(* Logix 5000 project; controller Uidaho_Factory vendor 1 type 14 code 165 rev 38.11; software revision 38.00; part 4 of 4 *)
(* tags used below, declared in another part *)
   MPO_Done : BOOL;
   MPO_Homing : BOOL;
   MPO_Oven_Start : BOOL;
   MPO_Turntable_Start : BOOL;
   SLD_Blue_Min : DINT;
   SLD_Blue_Time : DINT;
   SLD_Min_Value : DINT;
   SLD_Move_Time : DINT;
   SLD_Normal : DINT;
   SLD_Red_Min : DINT;
   SLD_Red_Time : DINT;
   SLD_start : DINT;
   SLD_Step : DINT;
   SLD_White_Time : DINT;
   Start : DINT;
   Step : DINT[20];
   StepTimers : TIMER[20];
   TurntableTimers : TIMER[10];
   VGR_HBW_Horizontal : DINT;   // The horizontal Encoder value for interfacing with HBW
   VGR_HBW_Rotate : DINT;
   VGR_HBW_Vertical : DINT;   // The Vertical Encoder value for interfacing with the HBW
   VGR_Horizontal_Target : DINT;
   VGR_Move_Horizontal : DINT;   // The horizontal encoder value for movement
   VGR_Move_Vertical : DINT;   // The vertical encoder value for movement
   VGR_MPO_Horizontal : DINT;   // The Horizontal encoderr value for interfacing with MPO
   VGR_MPO_Rotate : DINT;
   VGR_MPO_Vertical : DINT;   // The vertical encoder value for interfacing with MPO
   VGR_Rotation_Target : DINT;
   VGR_start : DINT;
   VGR_Step : DINT;
   VGR_Vertical_Target : DINT;
   Encoder_Counters_1X : COUNTER[10];
   PWM_Outputs : PWM_Out[20];
   Scaled_Analog_Color_Sensor_SLD : DINT;   // SLD - A1 = Color sensor
   VGR_PWM_Outputs : PWM_Out[20];
(* MainProgram, continued *)

ROUTINE MPO_Turntable_Process   (* ladder *)
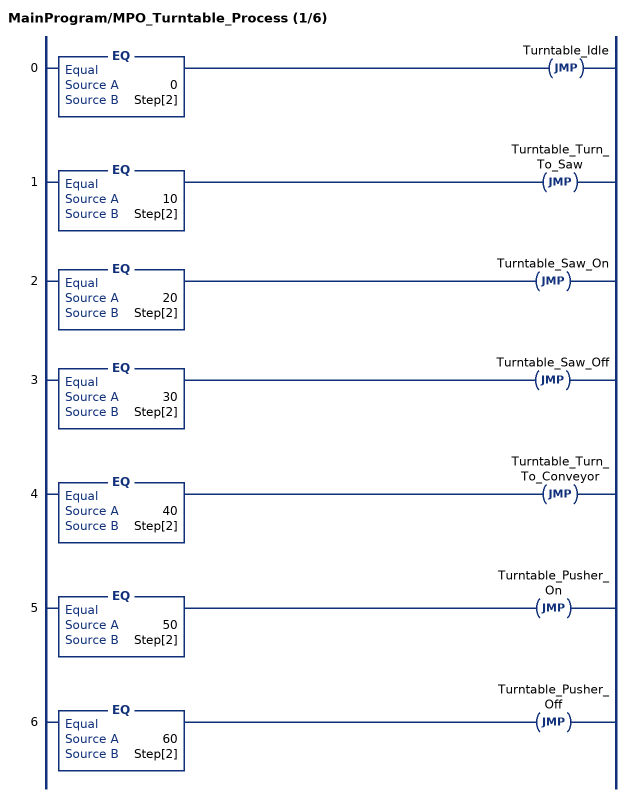
   0: EQ(0,Step[2])JMP(Turntable_Idle);
   1: EQ(10,Step[2])JMP(Turntable_Turn_To_Saw);
   2: EQ(20,Step[2])JMP(Turntable_Saw_On);
   3: EQ(30,Step[2])JMP(Turntable_Saw_Off);
   4: EQ(40,Step[2])JMP(Turntable_Turn_To_Conveyor);
   5: EQ(50,Step[2])JMP(Turntable_Pusher_On);
   6: EQ(60,Step[2])JMP(Turntable_Pusher_Off);
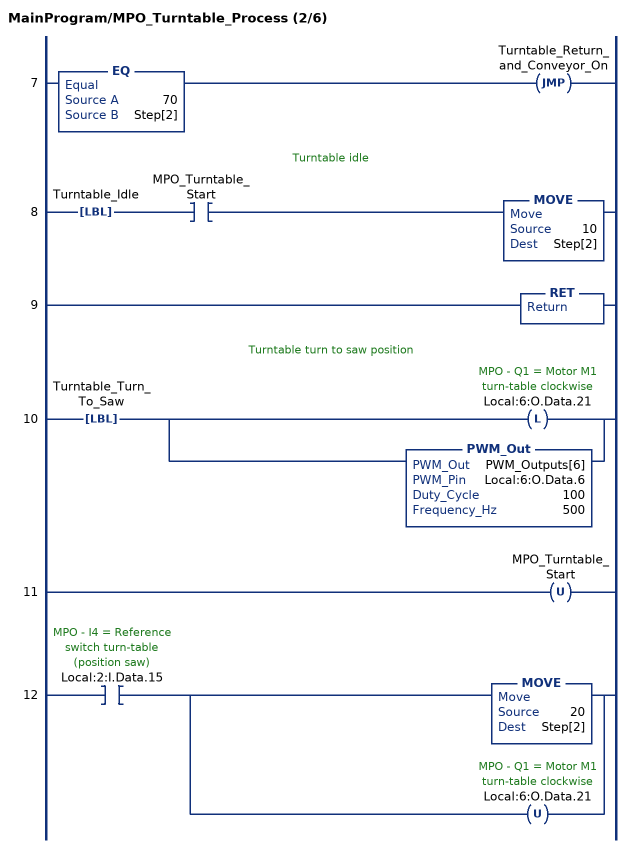
   7: EQ(70,Step[2])JMP(Turntable_Return_and_Conveyor_On);
   // Turntable idle
   8: LBL(Turntable_Idle)XIC(MPO_Turntable_Start)MOVE(10,Step[2]);
   9: RET();
   // Turntable turn to saw position
   10: LBL(Turntable_Turn_To_Saw)[OTL(Local:6:O.Data.21) ,PWM_Out(PWM_Outputs[6],Local:6:O.Data.6,100,500) ];
   11: OTU(MPO_Turntable_Start);
   12: XIC(Local:2:I.Data.15)[MOVE(20,Step[2]) ,OTU(Local:6:O.Data.21) ];
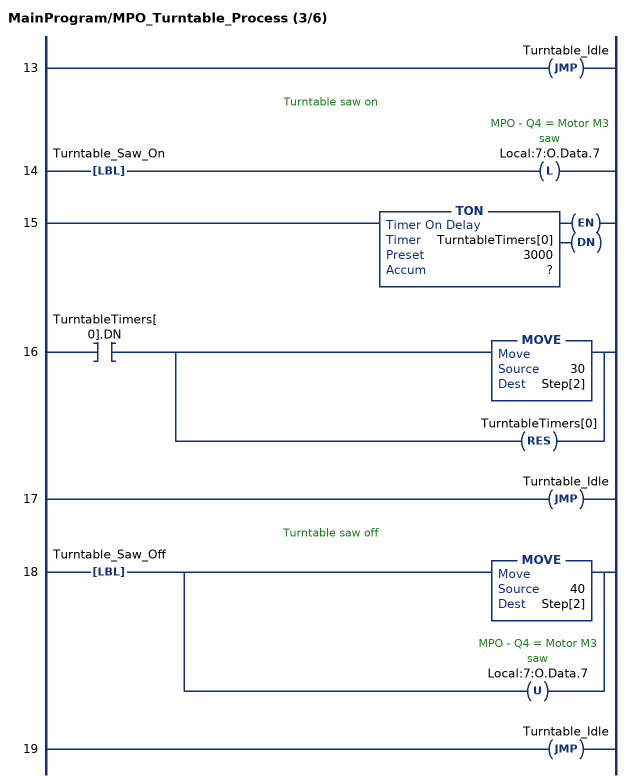
   13: JMP(Turntable_Idle);
   // Turntable saw on
   14: LBL(Turntable_Saw_On)OTL(Local:7:O.Data.7);
   15: TON(TurntableTimers[0],?,?);
   16: XIC(TurntableTimers[0].DN)[MOVE(30,Step[2]) ,RES(TurntableTimers[0]) ];
   17: JMP(Turntable_Idle);
   // Turntable saw off
   18: LBL(Turntable_Saw_Off)[MOVE(40,Step[2]) ,OTU(Local:7:O.Data.7) ];
   19: JMP(Turntable_Idle);
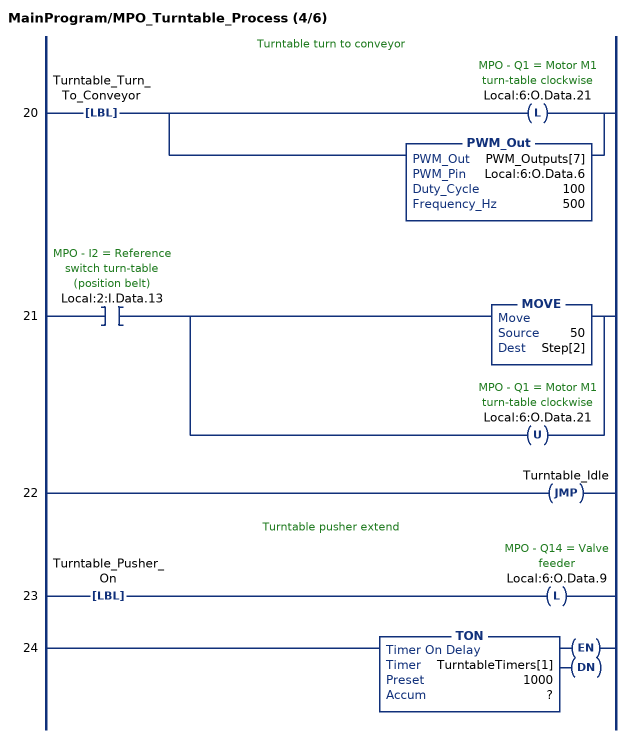
   // Turntable turn to conveyor
   20: LBL(Turntable_Turn_To_Conveyor)[OTL(Local:6:O.Data.21) ,PWM_Out(PWM_Outputs[7],Local:6:O.Data.6,100,500) ];
   21: XIC(Local:2:I.Data.13)[MOVE(50,Step[2]) ,OTU(Local:6:O.Data.21) ];
   22: JMP(Turntable_Idle);
   // Turntable pusher extend
   23: LBL(Turntable_Pusher_On)OTL(Local:6:O.Data.9);
   24: TON(TurntableTimers[1],?,?);
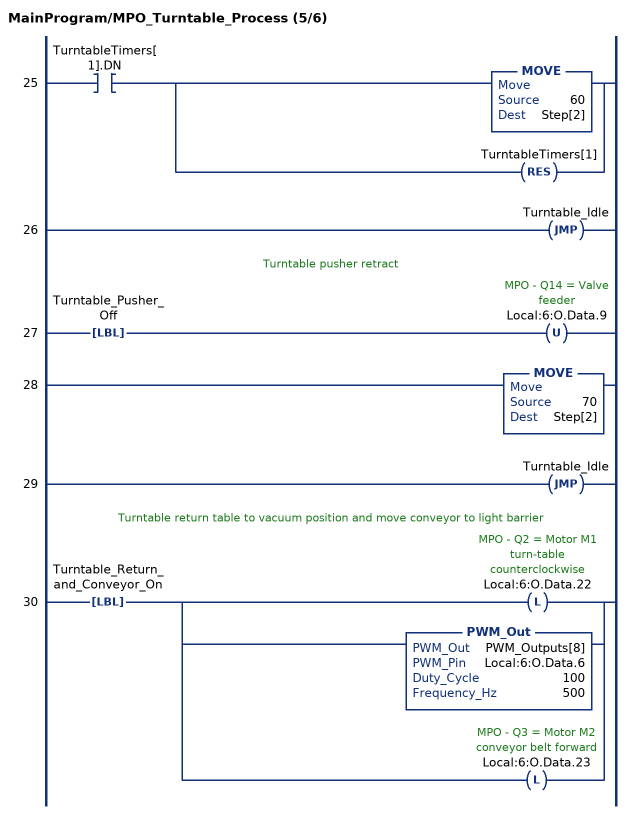
   25: XIC(TurntableTimers[1].DN)[MOVE(60,Step[2]) ,RES(TurntableTimers[1]) ];
   26: JMP(Turntable_Idle);
   // Turntable pusher retract
   27: LBL(Turntable_Pusher_Off)OTU(Local:6:O.Data.9);
   28: MOVE(70,Step[2]);
   29: JMP(Turntable_Idle);
   // Turntable return table to vacuum position and move conveyor to light barrier
   30: LBL(Turntable_Return_and_Conveyor_On)[[OTL(Local:6:O.Data.22) ,PWM_Out(PWM_Outputs[8],Local:6:O.Data.6,100,500) ] ,OTL(Local:6:O.Data.23) ];
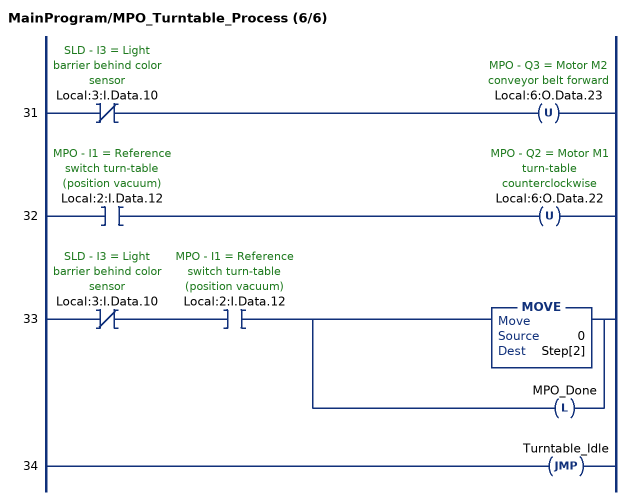
   31: XIO(Local:3:I.Data.10)OTU(Local:6:O.Data.23);
   32: XIC(Local:2:I.Data.12)OTU(Local:6:O.Data.22);
   33: XIO(Local:3:I.Data.10)XIC(Local:2:I.Data.12)[MOVE(0,Step[2]) ,OTL(MPO_Done) ];
   34: JMP(Turntable_Idle);
END_ROUTINE

ROUTINE SLD_Controller   (* ladder *)
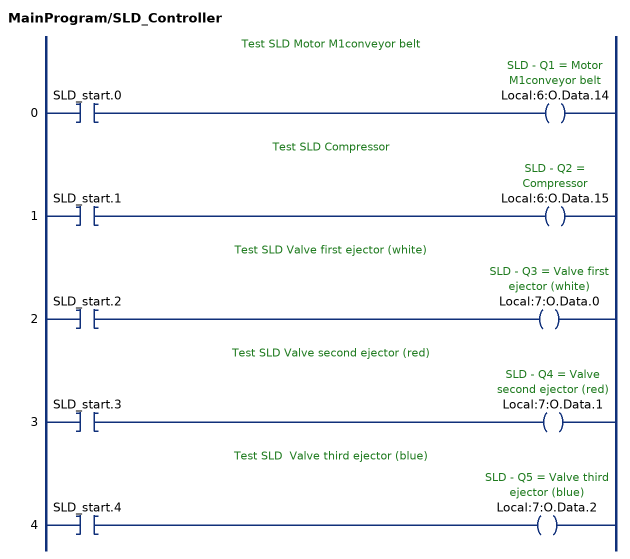
   // Test SLD Motor M1conveyor belt
   0: XIC(SLD_start.0)OTE(Local:6:O.Data.14);
   // Test SLD Compressor
   1: XIC(SLD_start.1)OTE(Local:6:O.Data.15);
   // Test SLD Valve first ejector (white)
   2: XIC(SLD_start.2)OTE(Local:7:O.Data.0);
   // Test SLD Valve second ejector (red)
   3: XIC(SLD_start.3)OTE(Local:7:O.Data.1);
   // Test SLD  Valve third ejector (blue)
   4: XIC(SLD_start.4)OTE(Local:7:O.Data.2);
END_ROUTINE

ROUTINE SLD_Sequencer   (* ladder *)
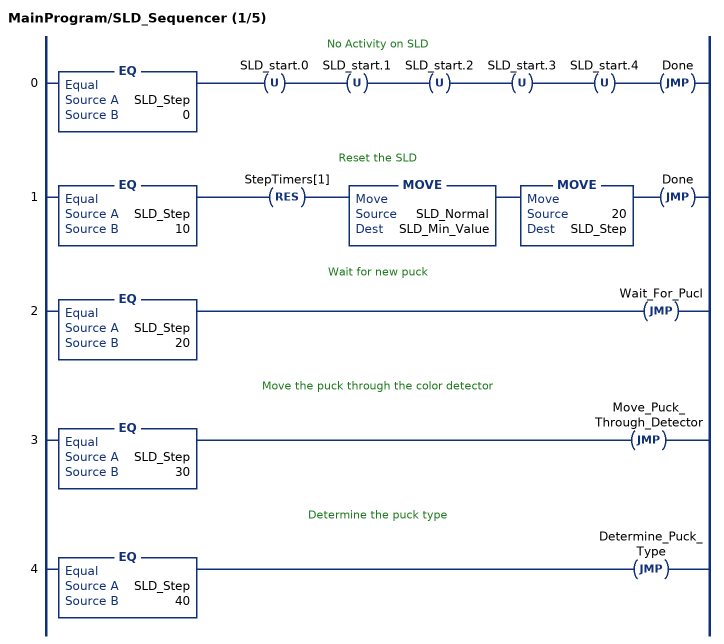
   // No Activity on SLD
   0: EQ(SLD_Step,0)OTU(SLD_start.0)OTU(SLD_start.1)OTU(SLD_start.2)OTU(SLD_start.3)OTU(SLD_start.4)JMP(Done);
   // Reset the SLD
   1: EQ(SLD_Step,10)RES(StepTimers[1])MOVE(SLD_Normal,SLD_Min_Value)MOVE(20,SLD_Step)JMP(Done);
   // Wait for new puck
   2: EQ(SLD_Step,20)JMP(Wait_For_Pucl);
   // Move the puck through the color detector
   3: EQ(SLD_Step,30)JMP(Move_Puck_Through_Detector);
   // Determine the puck type
   4: EQ(SLD_Step,40)JMP(Determine_Puck_Type);
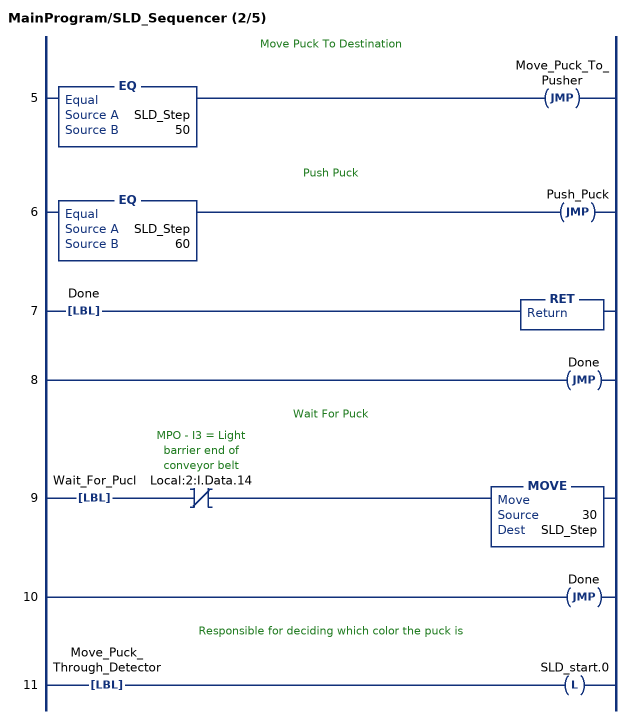
   // Move Puck To Destination
   5: EQ(SLD_Step,50)JMP(Move_Puck_To_Pusher);
   // Push Puck
   6: EQ(SLD_Step,60)JMP(Push_Puck);
   7: LBL(Done)RET();
   8: JMP(Done);
   // Wait For Puck
   9: LBL(Wait_For_Pucl)XIO(Local:2:I.Data.14)MOVE(30,SLD_Step);
   10: JMP(Done);
   // Responsible for deciding which color the puck is
   11: LBL(Move_Puck_Through_Detector)OTL(SLD_start.0);
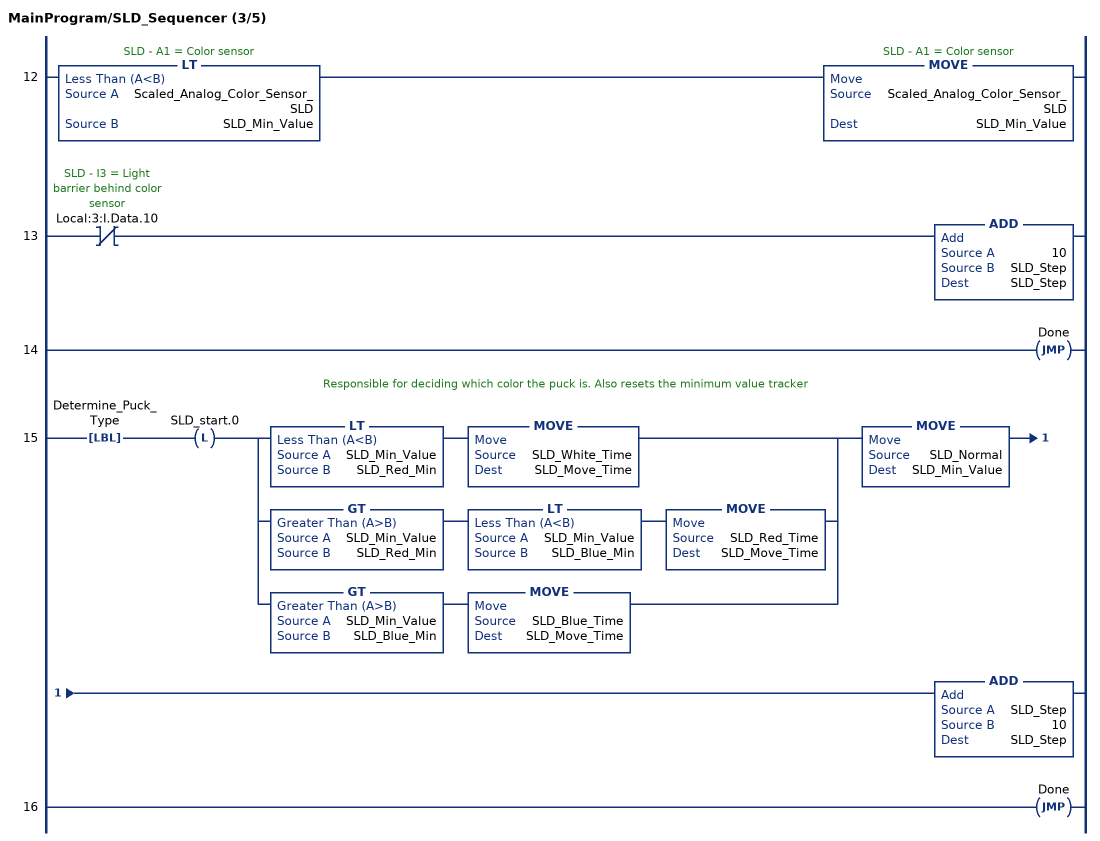
   12: LT(Scaled_Analog_Color_Sensor_SLD,SLD_Min_Value)MOVE(Scaled_Analog_Color_Sensor_SLD,SLD_Min_Value);
   13: XIO(Local:3:I.Data.10)ADD(10,SLD_Step,SLD_Step);
   14: JMP(Done);
   // Responsible for deciding which color the puck is. Also resets the minimum value tracker
   15: LBL(Determine_Puck_Type)OTL(SLD_start.0)[LT(SLD_Min_Value,SLD_Red_Min) MOVE(SLD_White_Time,SLD_Move_Time) ,GT(SLD_Min_Value,SLD_Red_Min) LT(SLD_Min_Value,SLD_Blue_Min) MOVE(SLD_Red_Time,SLD_Move_Time) ,GT(SLD_Min_Value,SLD_Blue_Min) MOVE(SLD_Blue_Time,SLD_Move_Time) ]MOVE(SLD_Normal,SLD_Min_Value)ADD(SLD_Step,10,SLD_Step);
   16: JMP(Done);
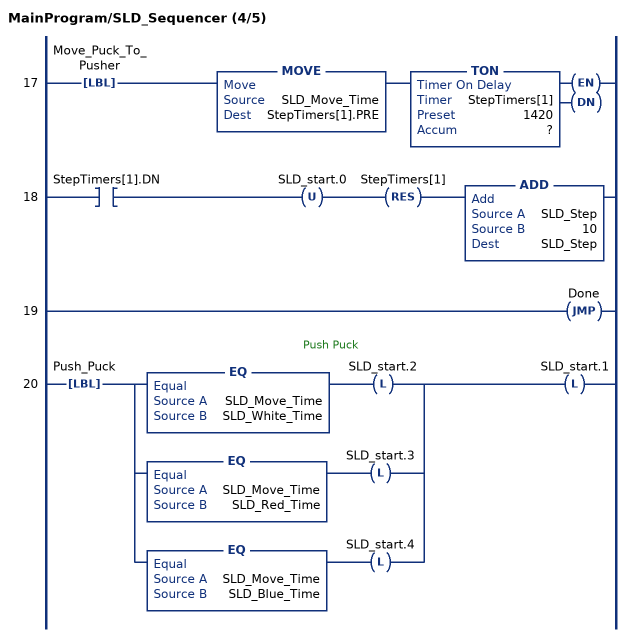
   17: LBL(Move_Puck_To_Pusher)MOVE(SLD_Move_Time,StepTimers[1].PRE)TON(StepTimers[1],?,?);
   18: XIC(StepTimers[1].DN)OTU(SLD_start.0)RES(StepTimers[1])ADD(SLD_Step,10,SLD_Step);
   19: JMP(Done);
   // Push Puck
   20: LBL(Push_Puck)[EQ(SLD_Move_Time,SLD_White_Time) OTL(SLD_start.2) ,EQ(SLD_Move_Time,SLD_Red_Time) OTL(SLD_start.3) ,EQ(SLD_Move_Time,SLD_Blue_Time) OTL(SLD_start.4) ]OTL(SLD_start.1);
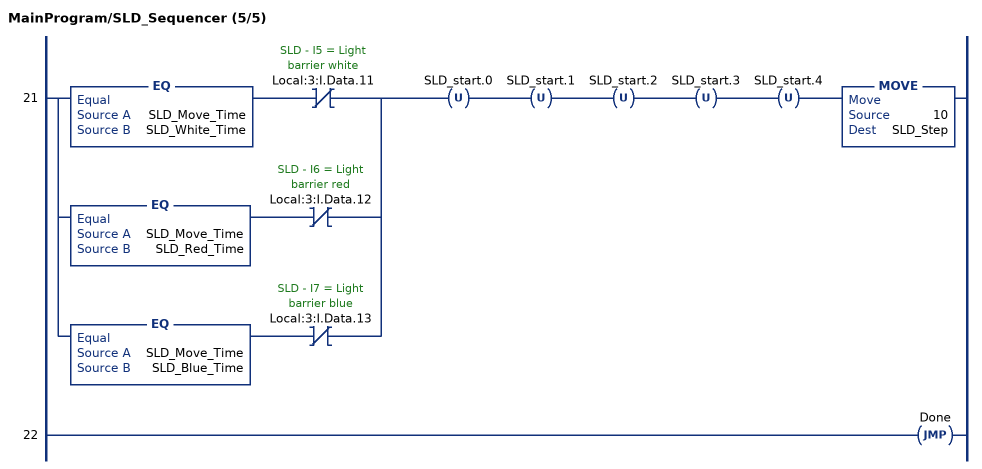
   21: [EQ(SLD_Move_Time,SLD_White_Time) XIO(Local:3:I.Data.11) ,EQ(SLD_Move_Time,SLD_Red_Time) XIO(Local:3:I.Data.12) ,EQ(SLD_Move_Time,SLD_Blue_Time) XIO(Local:3:I.Data.13) ]OTU(SLD_start.0)OTU(SLD_start.1)OTU(SLD_start.2)OTU(SLD_start.3)OTU(SLD_start.4)MOVE(10,SLD_Step);
   22: JMP(Done);
END_ROUTINE

ROUTINE VGR_Controller   (* ladder *)
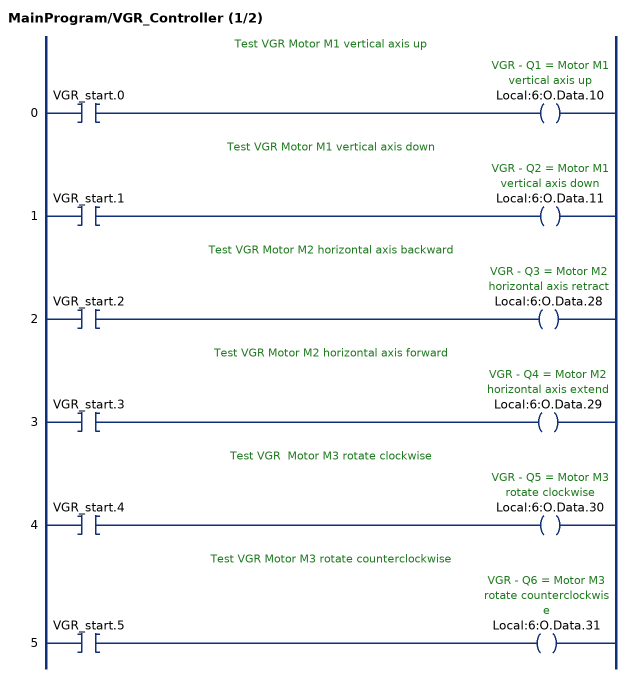
   // Test VGR Motor M1 vertical axis up
   0: XIC(VGR_start.0)OTE(Local:6:O.Data.10);
   // Test VGR Motor M1 vertical axis down
   1: XIC(VGR_start.1)OTE(Local:6:O.Data.11);
   // Test VGR Motor M2 horizontal axis backward
   2: XIC(VGR_start.2)OTE(Local:6:O.Data.28);
   // Test VGR Motor M2 horizontal axis forward
   3: XIC(VGR_start.3)OTE(Local:6:O.Data.29);
   // Test VGR  Motor M3 rotate clockwise
   4: XIC(VGR_start.4)OTE(Local:6:O.Data.30);
   // Test VGR Motor M3 rotate counterclockwise
   5: XIC(VGR_start.5)OTE(Local:6:O.Data.31);
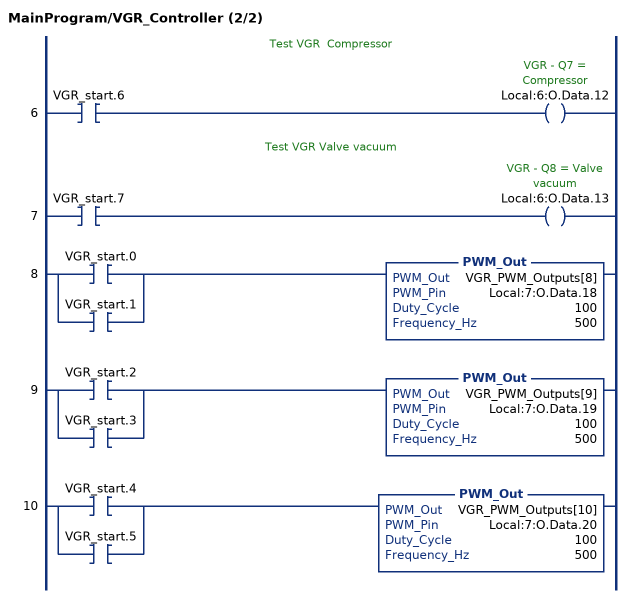
   // Test VGR  Compressor
   6: XIC(VGR_start.6)OTE(Local:6:O.Data.12);
   // Test VGR Valve vacuum
   7: XIC(VGR_start.7)OTE(Local:6:O.Data.13);
   8: [XIC(VGR_start.0) ,XIC(VGR_start.1) ]PWM_Out(VGR_PWM_Outputs[8],Local:7:O.Data.18,100,500);
   9: [XIC(VGR_start.2) ,XIC(VGR_start.3) ]PWM_Out(VGR_PWM_Outputs[9],Local:7:O.Data.19,100,500);
   10: [XIC(VGR_start.4) ,XIC(VGR_start.5) ]PWM_Out(VGR_PWM_Outputs[10],Local:7:O.Data.20,100,500);
END_ROUTINE

ROUTINE VGR_Sequencer   (* ladder *)
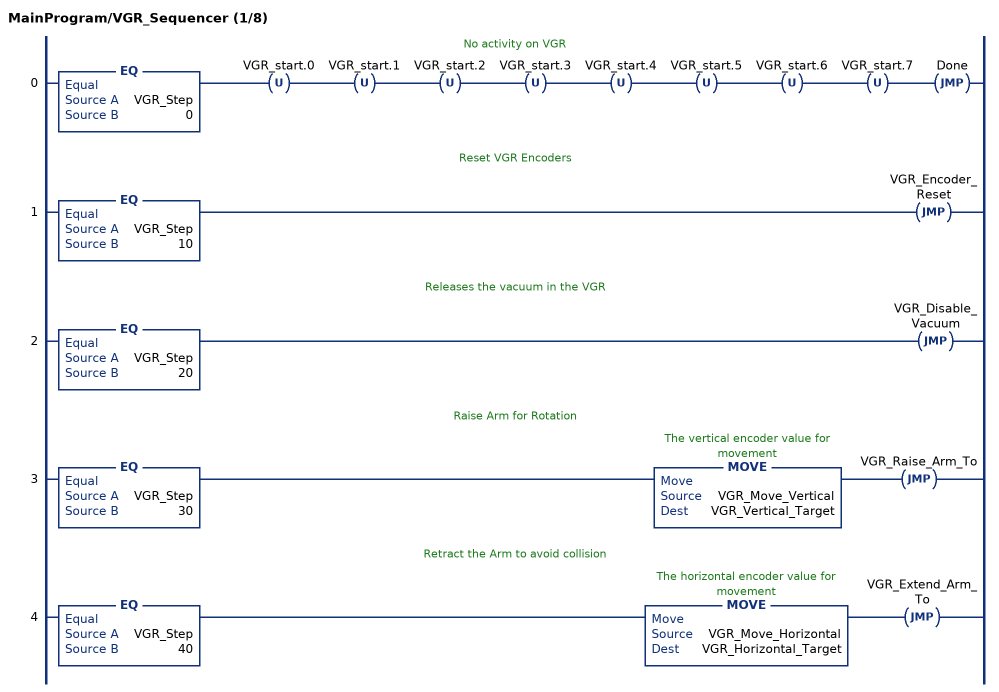
   // No activity on VGR
   0: EQ(VGR_Step,0)OTU(VGR_start.0)OTU(VGR_start.1)OTU(VGR_start.2)OTU(VGR_start.3)OTU(VGR_start.4)OTU(VGR_start.5)OTU(VGR_start.6)OTU(VGR_start.7)JMP(Done);
   // Reset VGR Encoders
   1: EQ(VGR_Step,10)JMP(VGR_Encoder_Reset);
   // Releases the vacuum in the VGR
   2: EQ(VGR_Step,20)JMP(VGR_Disable_Vacuum);
   // Raise Arm for Rotation
   3: EQ(VGR_Step,30)MOVE(VGR_Move_Vertical,VGR_Vertical_Target)JMP(VGR_Raise_Arm_To);
   // Retract the Arm to avoid collision
   4: EQ(VGR_Step,40)MOVE(VGR_Move_Horizontal,VGR_Horizontal_Target)JMP(VGR_Extend_Arm_To);
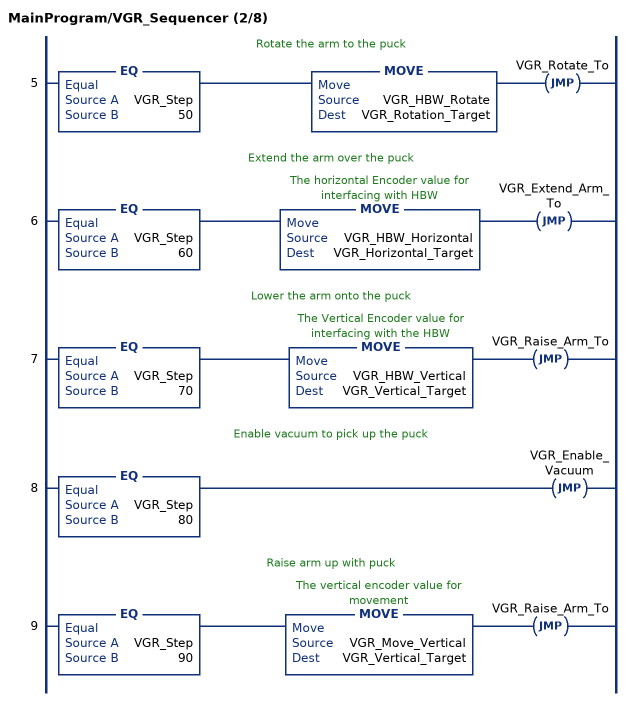
   // Rotate the arm to the puck
   5: EQ(VGR_Step,50)MOVE(VGR_HBW_Rotate,VGR_Rotation_Target)JMP(VGR_Rotate_To);
   // Extend the arm over the puck
   6: EQ(VGR_Step,60)MOVE(VGR_HBW_Horizontal,VGR_Horizontal_Target)JMP(VGR_Extend_Arm_To);
   // Lower the arm onto the puck
   7: EQ(VGR_Step,70)MOVE(VGR_HBW_Vertical,VGR_Vertical_Target)JMP(VGR_Raise_Arm_To);
   // Enable vacuum to pick up the puck
   8: EQ(VGR_Step,80)JMP(VGR_Enable_Vacuum);
   // Raise arm up with puck
   9: EQ(VGR_Step,90)MOVE(VGR_Move_Vertical,VGR_Vertical_Target)JMP(VGR_Raise_Arm_To);
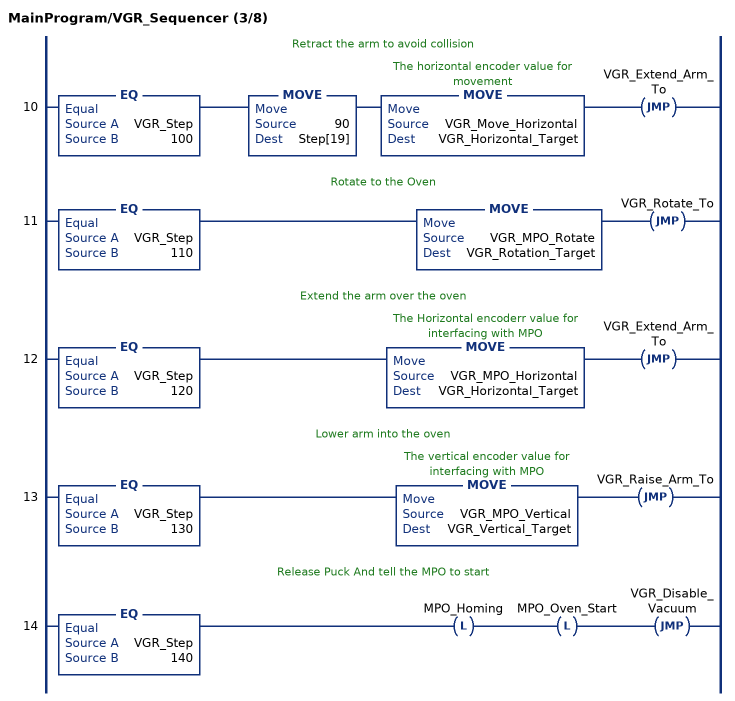
   // Retract the arm to avoid collision
   10: EQ(VGR_Step,100)MOVE(90,Step[19])MOVE(VGR_Move_Horizontal,VGR_Horizontal_Target)JMP(VGR_Extend_Arm_To);
   // Rotate to the Oven
   11: EQ(VGR_Step,110)MOVE(VGR_MPO_Rotate,VGR_Rotation_Target)JMP(VGR_Rotate_To);
   // Extend the arm over the oven
   12: EQ(VGR_Step,120)MOVE(VGR_MPO_Horizontal,VGR_Horizontal_Target)JMP(VGR_Extend_Arm_To);
   // Lower arm into the oven
   13: EQ(VGR_Step,130)MOVE(VGR_MPO_Vertical,VGR_Vertical_Target)JMP(VGR_Raise_Arm_To);
   // Release Puck And tell the MPO to start
   14: EQ(VGR_Step,140)OTL(MPO_Homing)OTL(MPO_Oven_Start)JMP(VGR_Disable_Vacuum);
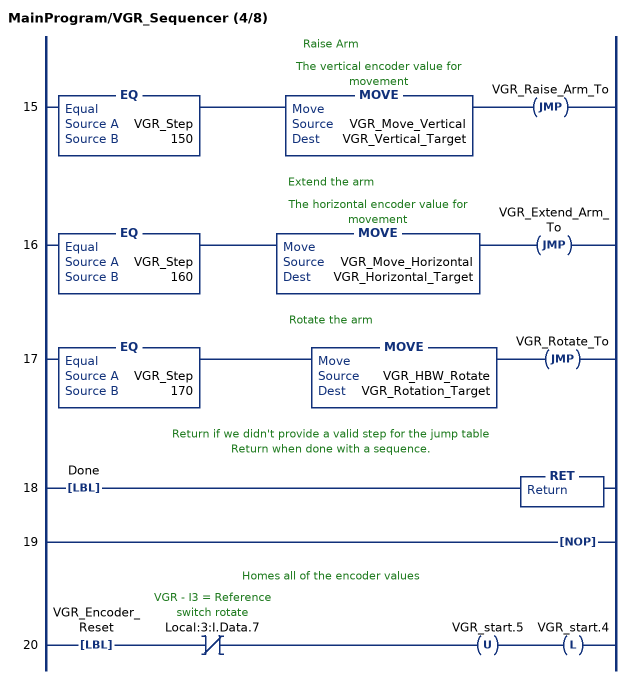
   // Raise Arm
   15: EQ(VGR_Step,150)MOVE(VGR_Move_Vertical,VGR_Vertical_Target)JMP(VGR_Raise_Arm_To);
   // Extend the arm
   16: EQ(VGR_Step,160)MOVE(VGR_Move_Horizontal,VGR_Horizontal_Target)JMP(VGR_Extend_Arm_To);
   // Rotate the arm
   17: EQ(VGR_Step,170)MOVE(VGR_HBW_Rotate,VGR_Rotation_Target)JMP(VGR_Rotate_To);
   // Return if we didn't provide a valid step for the jump table
   // Return when done with a sequence.
   18: LBL(Done)RET();
   19: NOP();
   // Homes all of the encoder values
   20: LBL(VGR_Encoder_Reset)XIO(Local:3:I.Data.7)OTU(VGR_start.5)OTL(VGR_start.4);
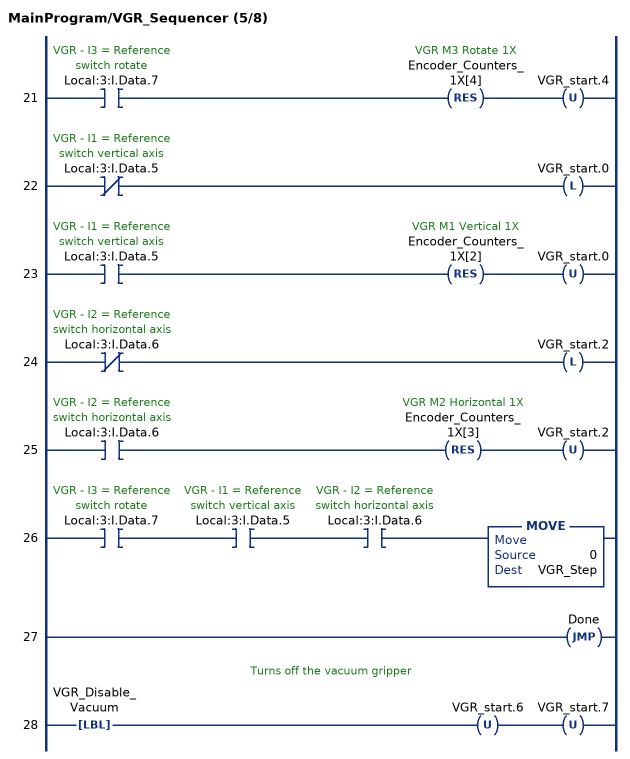
   21: XIC(Local:3:I.Data.7)RES(Encoder_Counters_1X[4])OTU(VGR_start.4);
   22: XIO(Local:3:I.Data.5)OTL(VGR_start.0);
   23: XIC(Local:3:I.Data.5)RES(Encoder_Counters_1X[2])OTU(VGR_start.0);
   24: XIO(Local:3:I.Data.6)OTL(VGR_start.2);
   25: XIC(Local:3:I.Data.6)RES(Encoder_Counters_1X[3])OTU(VGR_start.2);
   26: XIC(Local:3:I.Data.7)XIC(Local:3:I.Data.5)XIC(Local:3:I.Data.6)MOVE(0,VGR_Step);
   27: JMP(Done);
   // Turns off the vacuum gripper
   28: LBL(VGR_Disable_Vacuum)OTU(VGR_start.6)OTU(VGR_start.7);
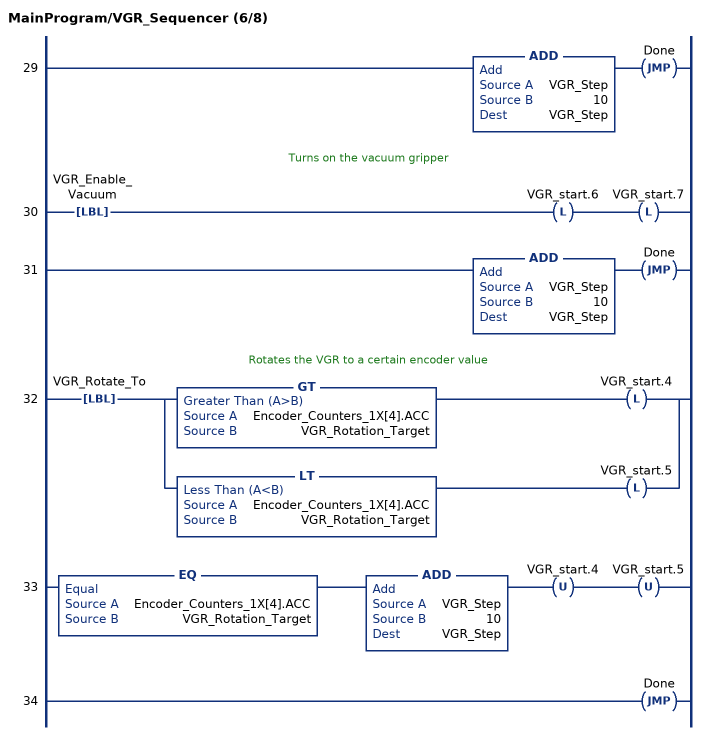
   29: ADD(VGR_Step,10,VGR_Step)JMP(Done);
   // Turns on the vacuum gripper
   30: LBL(VGR_Enable_Vacuum)OTL(VGR_start.6)OTL(VGR_start.7);
   31: ADD(VGR_Step,10,VGR_Step)JMP(Done);
   // Rotates the VGR to a certain encoder value
   32: LBL(VGR_Rotate_To)[GT(Encoder_Counters_1X[4].ACC,VGR_Rotation_Target) OTL(VGR_start.4) ,LT(Encoder_Counters_1X[4].ACC,VGR_Rotation_Target) OTL(VGR_start.5) ];
   33: EQ(Encoder_Counters_1X[4].ACC,VGR_Rotation_Target)ADD(VGR_Step,10,VGR_Step)OTU(VGR_start.4)OTU(VGR_start.5);
   34: JMP(Done);
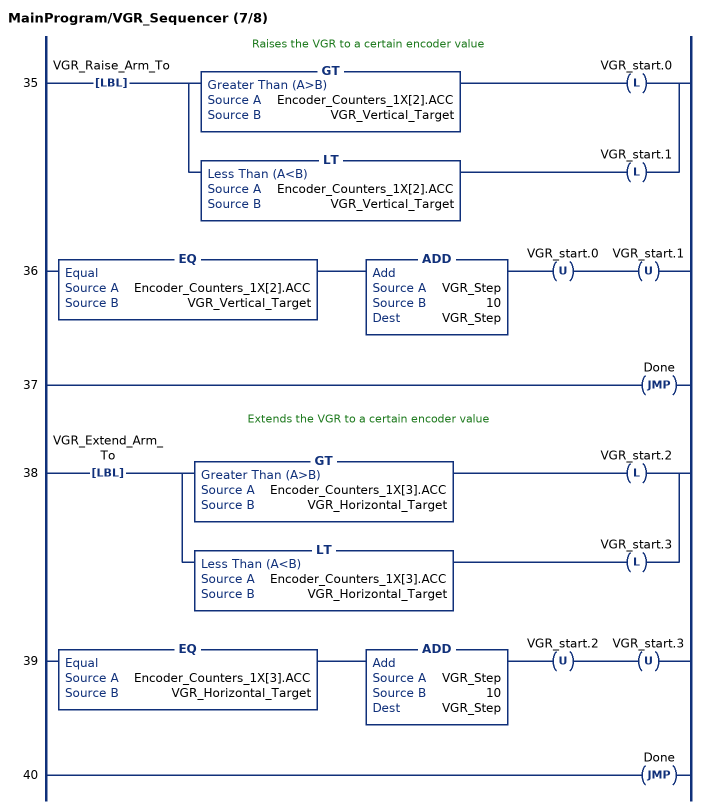
   // Raises the VGR to a certain encoder value
   35: LBL(VGR_Raise_Arm_To)[GT(Encoder_Counters_1X[2].ACC,VGR_Vertical_Target) OTL(VGR_start.0) ,LT(Encoder_Counters_1X[2].ACC,VGR_Vertical_Target) OTL(VGR_start.1) ];
   36: EQ(Encoder_Counters_1X[2].ACC,VGR_Vertical_Target)ADD(VGR_Step,10,VGR_Step)OTU(VGR_start.0)OTU(VGR_start.1);
   37: JMP(Done);
   // Extends the VGR to a certain encoder value
   38: LBL(VGR_Extend_Arm_To)[GT(Encoder_Counters_1X[3].ACC,VGR_Horizontal_Target) OTL(VGR_start.2) ,LT(Encoder_Counters_1X[3].ACC,VGR_Horizontal_Target) OTL(VGR_start.3) ];
   39: EQ(Encoder_Counters_1X[3].ACC,VGR_Horizontal_Target)ADD(VGR_Step,10,VGR_Step)OTU(VGR_start.2)OTU(VGR_start.3);
   40: JMP(Done);
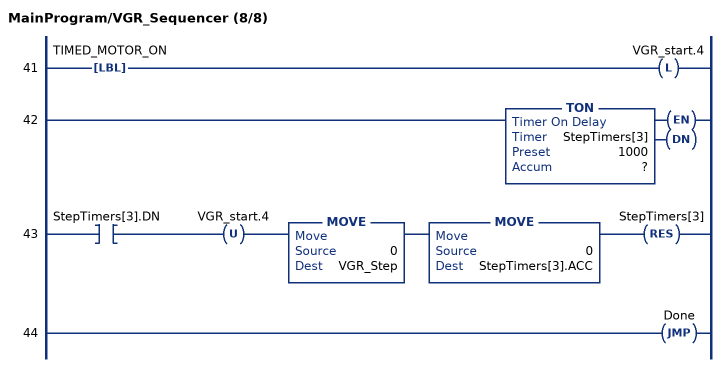
   41: LBL(TIMED_MOTOR_ON)OTL(VGR_start.4);
   42: TON(StepTimers[3],?,?);
   43: XIC(StepTimers[3].DN)OTU(VGR_start.4)MOVE(0,VGR_Step)MOVE(0,StepTimers[3].ACC)RES(StepTimers[3]);
   44: JMP(Done);
END_ROUTINE
END_PROGRAM
